VAR_GLOBAL	
	
	// DINT inputs
	n_pS : REAL;
	n_pR : REAL;
	n_pCB : REAL;
	n_pCA : REAL;
	n_pWA1 : REAL;
	n_pWB1 : REAL;
	n_pWA: REAL;
	n_pWB : REAL;
	n_pWD : REAL;
	n_QW : REAL;
	n_Xc : REAL;
	n_JoyX : REAL;
	n_JoyY : REAL;
	n_WinchEncoder : REAL;
	
END_VAR

(* stored: Version 1.1.0.1, ProductVersion 3.1.4024.12
   GVL G_HMI: Id {189070c1-188a-4360-bbe2-0d9f5ef44910} *)
